% RSLogix 500 project CONTROL_BAK113.RSS, saved by version 7.30.00.17 %
PROJECT "UNTITLED"    % processor: MicroLogix 1500 %

PROGRAM FILES
  LAD 2 "PRINCIPAL"  4 rungs
  LAD 3 "FLUJO"  6 rungs
  LAD 4 "NIVEL"  9 rungs
  LAD 5 "BOMBAS"  33 rungs

DATA FILES
  O0 OUTPUT  41 elements
  I1 INPUT  59 elements
  S2 STATUS  66 elements
  B3 BINARY  1 elements
  T4 TIMER  1 elements
  C5 COUNTER  1 elements
  R6 CONTROL  1 elements
  N7 INTEGER  25 elements
  F8 FLOAT  23 elements
  PD9   2 elements

LADDER 2 "PRINCIPAL"
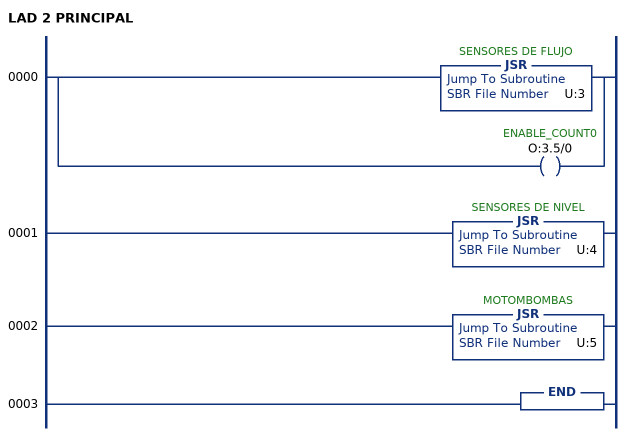
% Rung: 0 %
SOR BST JSR U:3 NXB OTE O:3.5/0 BND EOR
%   U:3  "SENSORES DE FLUJO" %
%   O:3.5/0  ENABLE_COUNT0 %
% Rung: 1 %
SOR JSR U:4 EOR
%   U:4  "SENSORES DE NIVEL" %
% Rung: 2 %
SOR JSR U:5 EOR
%   U:5  "MOTOMBOMBAS" %
% Rung: 3 %
SOR END EOR

LADDER 3 "FLUJO"
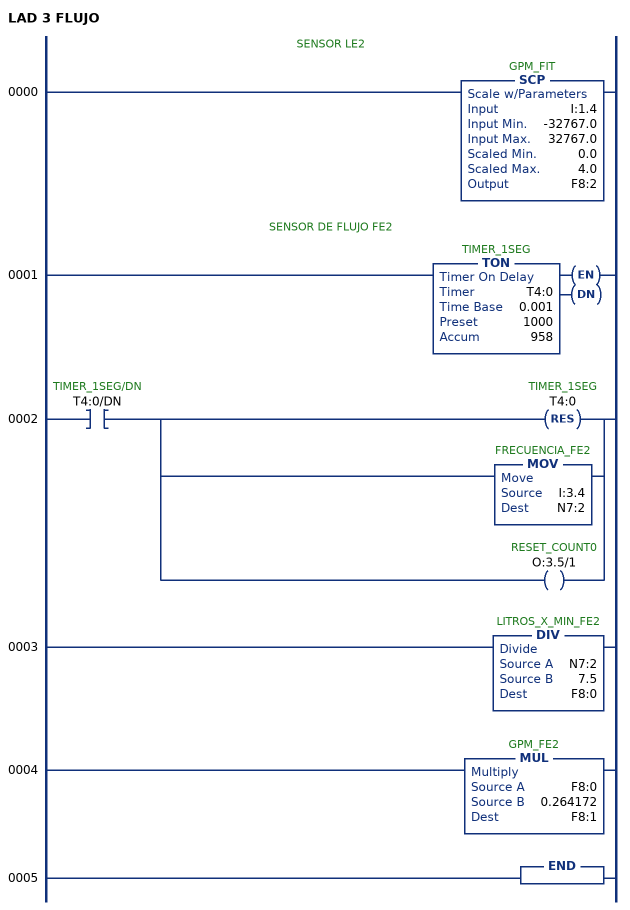
% Rung: 0 %
% SENSOR LE2 %
SOR SCP I:1.4 -32767.0 32767.0 0.0 4.0 F8:2 EOR
%   I:1.4  TRANSMISOR_FIT %
%   F8:2  GPM_FIT %
% Rung: 1 %
% SENSOR DE FLUJO FE2 %
SOR TON T4:0 0.001 1000 958 EOR
%   T4:0  TIMER_1SEG %
% Rung: 2 %
SOR XIC T4:0/DN BST RES T4:0 NXB MOV I:3.4 N7:2 NXB OTE O:3.5/1 BND EOR
%   T4:0  TIMER_1SEG %
%   N7:2  FRECUENCIA_FE2 %
%   O:3.5/1  RESET_COUNT0 %
% Rung: 3 %
SOR DIV N7:2 7.5 F8:0 EOR
%   N7:2  FRECUENCIA_FE2 %
%   F8:0  LITROS_X_MIN_FE2 %
% Rung: 4 %
SOR MUL F8:0 0.264172 F8:1 EOR
%   F8:0  LITROS_X_MIN_FE2 %
%   F8:1  GPM_FE2 %
% Rung: 5 %
SOR END EOR

LADDER 4 "NIVEL"
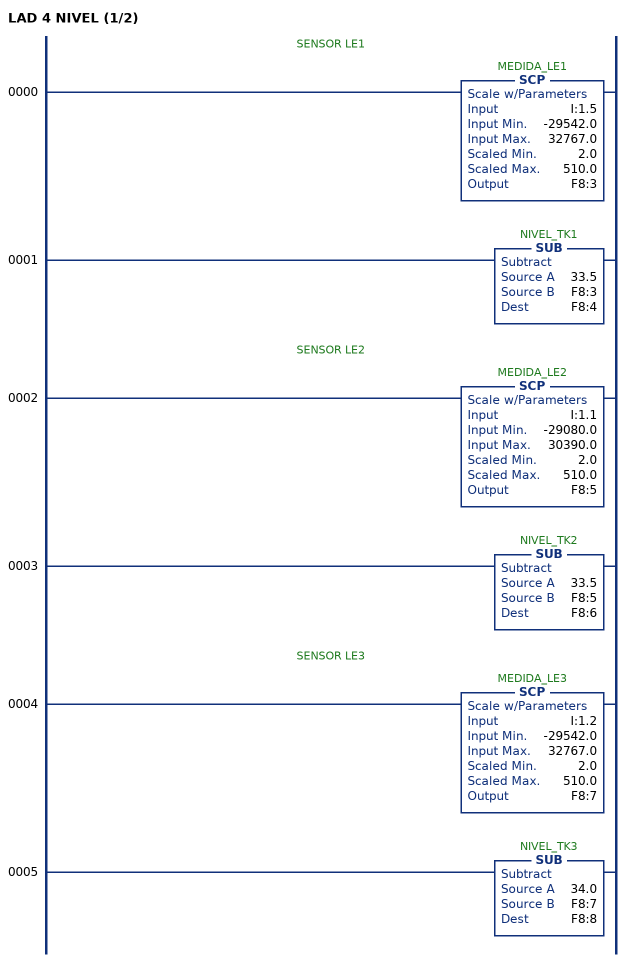
% Rung: 0 %
% SENSOR LE1 %
SOR SCP I:1.5 -29542.0 32767.0 2.0 510.0 F8:3 EOR
%   F8:3  MEDIDA_LE1 %
% Rung: 1 %
SOR SUB 33.5 F8:3 F8:4 EOR
%   F8:3  MEDIDA_LE1 %
%   F8:4  NIVEL_TK1 %
% Rung: 2 %
% SENSOR LE2 %
SOR SCP I:1.1 -29080.0 30390.0 2.0 510.0 F8:5 EOR
%   I:1.1  LE2 %
%   F8:5  MEDIDA_LE2 %
% Rung: 3 %
SOR SUB 33.5 F8:5 F8:6 EOR
%   F8:5  MEDIDA_LE2 %
%   F8:6  NIVEL_TK2 %
% Rung: 4 %
% SENSOR LE3 %
SOR SCP I:1.2 -29542.0 32767.0 2.0 510.0 F8:7 EOR
%   I:1.2  LE3 %
%   F8:7  MEDIDA_LE3 %
% Rung: 5 %
SOR SUB 34.0 F8:7 F8:8 EOR
%   F8:7  MEDIDA_LE3 %
%   F8:8  NIVEL_TK3 %

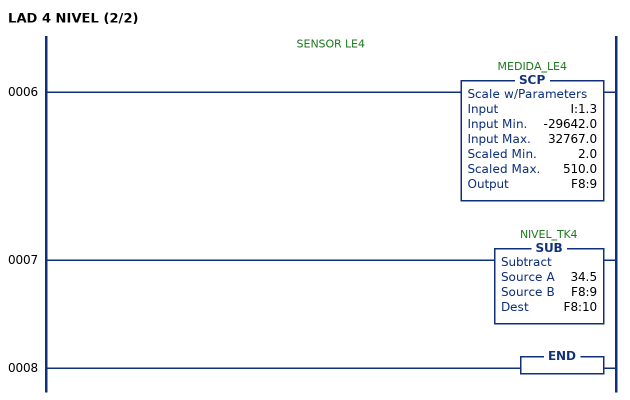
% Rung: 6 %
% SENSOR LE4 %
SOR SCP I:1.3 -29642.0 32767.0 2.0 510.0 F8:9 EOR
%   I:1.3  LE4 %
%   F8:9  MEDIDA_LE4 %
% Rung: 7 %
SOR SUB 34.5 F8:9 F8:10 EOR
%   F8:9  MEDIDA_LE4 %
%   F8:10  NIVEL_TK4 %
% Rung: 8 %
SOR END EOR

LADDER 5 "BOMBAS"
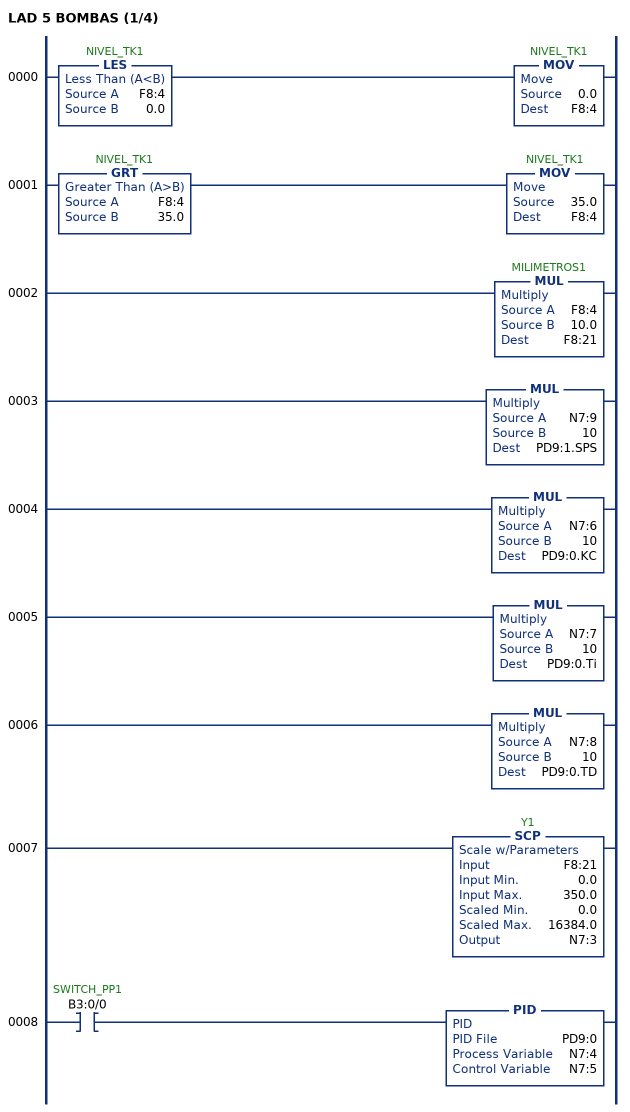
% Rung: 0 %
SOR LES F8:4 0.0 MOV 0.0 F8:4 EOR
%   F8:4  NIVEL_TK1 %
% Rung: 1 %
SOR GRT F8:4 35.0 MOV 35.0 F8:4 EOR
%   F8:4  NIVEL_TK1 %
% Rung: 2 %
SOR MUL F8:4 10.0 F8:21 EOR
%   F8:4  NIVEL_TK1 %
%   F8:21  MILIMETROS1 %
% Rung: 3 %
SOR MUL N7:9 10 PD9:1.SPS EOR
%   N7:9  N %
% Rung: 4 %
SOR MUL N7:6 10 PD9:0.KC EOR
% Rung: 5 %
SOR MUL N7:7 10 PD9:0.Ti EOR
% Rung: 6 %
SOR MUL N7:8 10 PD9:0.TD EOR
% Rung: 7 %
SOR SCP F8:21 0.0 350.0 0.0 16384.0 N7:3 EOR
%   F8:21  MILIMETROS1 %
%   N7:3  Y1 %
% Rung: 8 %
SOR XIC B3:0/0 PID PD9:0 N7:4 N7:5 EOR
%   B3:0/0  SWITCH_PP1 %
%   N7:4  Y2 %
%   N7:5  PID1 %

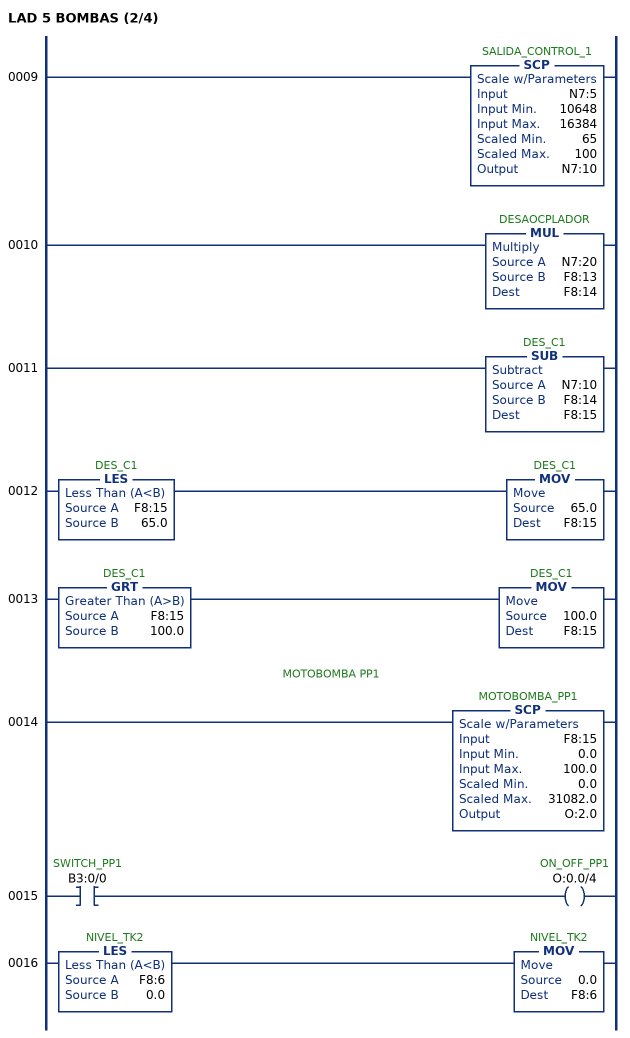
% Rung: 9 %
SOR SCP N7:5 10648 16384 65 100 N7:10 EOR
%   N7:5  PID1 %
%   N7:10  SALIDA_CONTROL_1 %
% Rung: 10 %
SOR MUL N7:20 F8:13 F8:14 EOR
%   N7:20  SALIDA_CONTROL_2 %
%   F8:13  D12 %
%   F8:14  DESAOCPLADOR %
% Rung: 11 %
SOR SUB N7:10 F8:14 F8:15 EOR
%   N7:10  SALIDA_CONTROL_1 %
%   F8:14  DESAOCPLADOR %
%   F8:15  DES_C1 %
% Rung: 12 %
SOR LES F8:15 65.0 MOV 65.0 F8:15 EOR
%   F8:15  DES_C1 %
% Rung: 13 %
SOR GRT F8:15 100.0 MOV 100.0 F8:15 EOR
%   F8:15  DES_C1 %
% Rung: 14 %
% MOTOBOMBA PP1 %
SOR SCP F8:15 0.0 100.0 0.0 31082.0 O:2.0 EOR
%   F8:15  DES_C1 %
%   O:2.0  MOTOBOMBA_PP1 %
% Rung: 15 %
SOR XIC B3:0/0 OTE O:0.0/4 EOR
%   B3:0/0  SWITCH_PP1 %
%   O:0.0/4  ON_OFF_PP1 %
% Rung: 16 %
SOR LES F8:6 0.0 MOV 0.0 F8:6 EOR
%   F8:6  NIVEL_TK2 %

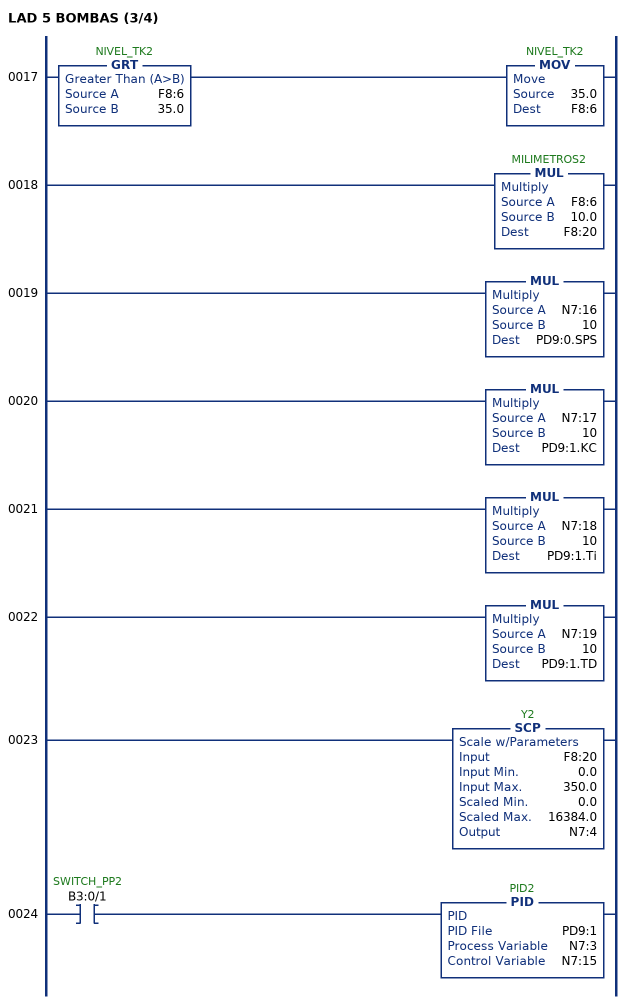
% Rung: 17 %
SOR GRT F8:6 35.0 MOV 35.0 F8:6 EOR
%   F8:6  NIVEL_TK2 %
% Rung: 18 %
SOR MUL F8:6 10.0 F8:20 EOR
%   F8:6  NIVEL_TK2 %
%   F8:20  MILIMETROS2 %
% Rung: 19 %
SOR MUL N7:16 10 PD9:0.SPS EOR
% Rung: 20 %
SOR MUL N7:17 10 PD9:1.KC EOR
% Rung: 21 %
SOR MUL N7:18 10 PD9:1.Ti EOR
%   N7:18  TI2 %
% Rung: 22 %
SOR MUL N7:19 10 PD9:1.TD EOR
%   N7:19  TD2 %
% Rung: 23 %
SOR SCP F8:20 0.0 350.0 0.0 16384.0 N7:4 EOR
%   F8:20  MILIMETROS2 %
%   N7:4  Y2 %
% Rung: 24 %
SOR XIC B3:0/1 PID PD9:1 N7:3 N7:15 EOR
%   B3:0/1  SWITCH_PP2 %
%   PD9:1  PID2 %
%   N7:3  Y1 %

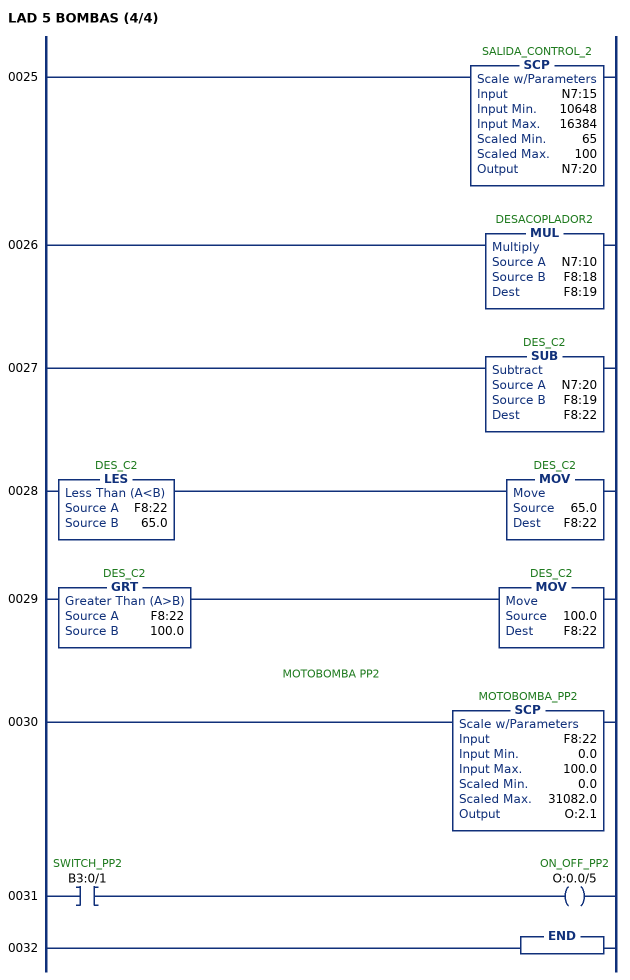
% Rung: 25 %
SOR SCP N7:15 10648 16384 65 100 N7:20 EOR
%   N7:20  SALIDA_CONTROL_2 %
% Rung: 26 %
SOR MUL N7:10 F8:18 F8:19 EOR
%   N7:10  SALIDA_CONTROL_1 %
%   F8:18  D22 %
%   F8:19  DESACOPLADOR2 %
% Rung: 27 %
SOR SUB N7:20 F8:19 F8:22 EOR
%   N7:20  SALIDA_CONTROL_2 %
%   F8:19  DESACOPLADOR2 %
%   F8:22  DES_C2 %
% Rung: 28 %
SOR LES F8:22 65.0 MOV 65.0 F8:22 EOR
%   F8:22  DES_C2 %
% Rung: 29 %
SOR GRT F8:22 100.0 MOV 100.0 F8:22 EOR
%   F8:22  DES_C2 %
% Rung: 30 %
% MOTOBOMBA PP2 %
SOR SCP F8:22 0.0 100.0 0.0 31082.0 O:2.1 EOR
%   F8:22  DES_C2 %
%   O:2.1  MOTOBOMBA_PP2 %
% Rung: 31 %
SOR XIC B3:0/1 OTE O:0.0/5 EOR
%   B3:0/1  SWITCH_PP2 %
%   O:0.0/5  ON_OFF_PP2 %
% Rung: 32 %
SOR END EOR

OTHER DOCUMENTED ADDRESSES
  F8:11  G12
  F8:12  G11
  F8:16  G21
  F8:17  G22
  I:1.0  LE1
  N7:0  FRECUENCIA_PP1
  N7:1  FRECUENCIA_PP2
  PD9:0.2  SP1
  PD9:0.3  KC1
  PD9:0.4  TI1
  PD9:0.5  TD1
  PD9:1.2  SP2
  PD9:1.3  KC2
  PD9:1.4  T12
  PD9:1.5  TD21

DATA TABLE (non-zero values as saved)
DATA T4
% .PRE .ACC %
% T4:0 % 1000 958
DATA N7
% N7:0 % 0 0 0 7250 4477 10648 2 263 66 15
% N7:10 % 65 15 0 0 0 10648 0 0 0 0
% N7:20 % 65 0 0 0 0
DATA F8
% F8:0 % 0 0 0 22.26815 11.23185
% F8:5 % 33.40939 0.09061432 32.22285 1.777145 31.71046
% F8:10 % 2.789541 0 0 0 0
% F8:15 % 50 0 0 0 0
